FUNCTION_BLOCK Valvula_Higienizacao_HMI (* Service Interface Function Block Type *)
  (* Standard: 61499-2 *)
  (* Version 0.0, 04/03/2026, template *)
  PACKAGE Hidryco.HidrycoLib;
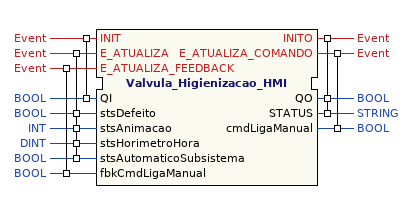
  EVENT_INPUT
    INIT WITH QI;
    E_ATUALIZA WITH stsDefeito, stsAnimacao, stsHorimetroHora, stsAutomaticoSubsistema;
    E_ATUALIZA_FEEDBACK WITH fbkCmdLigaManual;
  END_EVENT
  EVENT_OUTPUT
    INITO WITH QO, STATUS;
    E_ATUALIZA_COMANDO WITH cmdLigaManual;
  END_EVENT
  VAR_INPUT
    QI : BOOL;
    stsDefeito : BOOL;
    stsAnimacao : INT;
    stsHorimetroHora : DINT;
    stsAutomaticoSubsistema : BOOL;
    fbkCmdLigaManual : BOOL;
  END_VAR
  VAR_OUTPUT
    QO : BOOL; (* Event Output Qualifier *)
    STATUS : STRING; (* Service Status *)
    cmdLigaManual : BOOL;
  END_VAR
  SERVICE /
    SEQUENCE 
    END_SEQUENCE
  END_SERVICE
END_FUNCTION_BLOCK
